// TIA Portal V17 export
// export: Created 2026-04-13T11:12:45.2431947Z, ExportSetting WithDefaults, DisplayName Totally Integrated Automation Portal, DisplayVersion V17 Update 4, DisplayName TIA Portal Openness, DisplayVersion V17 Update 4, DisplayName TIA Portal Version Control Interface, DisplayVersion V17, DisplayName SINAMICS Startdrive Advanced, DisplayVersion V17, DisplayName SINAMICS Startdrive G130, G150, S120, S150, SINAMICS MV, S210, DisplayVersion V17, DisplayName SINAMICS Startdrive G110M, G120, G120C, G120D, G120P, G115D, DisplayVersion V17, DisplayName STEP 7 Professional, DisplayVersion V17 Update 4, DisplayName STEP 7 Safety, DisplayVersion V17, DisplayName WinCC Professional, DisplayVersion V17 Update 4
VAR_GLOBAL   // PLC tag table "IO"
   "I0.0" AT %I0.0 : Bool;
   "I0.1" AT %I0.1 : Bool;
   "I0.2" AT %I0.2 : Bool;
   "I0.3" AT %I0.3 : Bool;
   "I0.4" AT %I0.4 : Bool;
   "I0.5" AT %I0.5 : Bool;
   "I0.6" AT %I0.6 : Bool;
   "I0.7" AT %I0.7 : Bool;
   "I1.0" AT %I1.0 : Bool;
   "I1.1" AT %I1.1 : Bool;
   "I2.0" AT %I2.0 : Bool;
   "I2.1" AT %I2.1 : Bool;
   "I2.2" AT %I2.2 : Bool;
   "I2.3" AT %I2.3 : Bool;
   "I2.4" AT %I2.4 : Bool;
   "I2.5" AT %I2.5 : Bool;
   "I2.6" AT %I2.6 : Bool;
   "I2.7" AT %I2.7 : Bool;
   "I3.0" AT %I3.0 : Bool;
   "I3.1" AT %I3.1 : Bool;
   "I3.2" AT %I3.2 : Bool;
   "I3.3" AT %I3.3 : Bool;
   "I3.4" AT %I3.4 : Bool;
   "I3.5" AT %I3.5 : Bool;
   "I3.6" AT %I3.6 : Bool;
   "I3.7" AT %I3.7 : Bool;
   "I4.0" AT %I4.0 : Bool;
   "I4.1" AT %I4.1 : Bool;
   "I4.2" AT %I4.2 : Bool;
   "I4.3" AT %I4.3 : Bool;
   "I4.4" AT %I4.4 : Bool;
   "I4.5" AT %I4.5 : Bool;
   "I4.6" AT %I4.6 : Bool;
   "I4.7" AT %I4.7 : Bool;
   "I5.0" AT %I5.0 : Bool;
   "I5.1" AT %I5.1 : Bool;
   "I5.2" AT %I5.2 : Bool;
   "I5.3" AT %I5.3 : Bool;
   "I5.4" AT %I5.4 : Bool;
   "I5.5" AT %I5.5 : Bool;
   "I5.6" AT %I5.6 : Bool;
   "I5.7" AT %I5.7 : Bool;
   "Q0.1" AT %Q0.1 : Bool;
   "Q0.2" AT %Q0.2 : Bool;
   "Q0.3" AT %Q0.3 : Bool;
   "Q0.4" AT %Q0.4 : Bool;
   "Q0.5" AT %Q0.5 : Bool;
   "Q0.6" AT %Q0.6 : Bool;
   "Q0.7" AT %Q0.7 : Bool;
   "Q1.0" AT %Q1.0 : Bool;
   "Q1.1" AT %Q1.1 : Bool;
   "Q1.2" AT %Q1.2 : Bool;
   "Q1.3" AT %Q1.3 : Bool;
   "Q1.4" AT %Q1.4 : Bool;
   "Q1.5" AT %Q1.5 : Bool;
   "Q3.0" AT %Q3.0 : Bool;
   "Q3.1" AT %Q3.1 : Bool;
   "Q3.2" AT %Q3.2 : Bool;
   "Q3.3" AT %Q3.3 : Bool;
   "Q3.4" AT %Q3.4 : Bool;
   "Q3.5" AT %Q3.5 : Bool;
   "Q3.6" AT %Q3.6 : Bool;
   "Q3.7" AT %Q3.7 : Bool;
   "Q4.0" AT %Q4.0 : Bool;
   "Q4.1" AT %Q4.1 : Bool;
   "Q4.2" AT %Q4.2 : Bool;
   "Q4.3" AT %Q4.3 : Bool;
   "Q4.4" AT %Q4.4 : Bool;
   "Q4.5" AT %Q4.5 : Bool;
   "Q4.6" AT %Q4.6 : Bool;
   "Q4.7" AT %Q4.7 : Bool;
   "Q5.0" AT %Q5.0 : Bool;
   "Q5.1" AT %Q5.1 : Bool;
   "Q5.2" AT %Q5.2 : Bool;
   "Q5.3" AT %Q5.3 : Bool;
   "Q5.4" AT %Q5.4 : Bool;
   "Q0.0" AT %Q0.0 : Bool;
   "I1.2" AT %I1.2 : Bool;
   "I1.3" AT %I1.3 : Bool;
   "I1.4" AT %I1.4 : Bool;
   "I1.5" AT %I1.5 : Bool;
   "Q5.5" AT %Q5.5 : Bool;
   "Q1.6" AT %Q1.6 : Bool;
   "Q1.7" AT %Q1.7 : Bool;
   "I1.6" AT %I1.6 : Bool;
   "I1.7" AT %I1.7 : Bool;
   "Q5.6" AT %Q5.6 : Bool;
   "Q5.7" AT %Q5.7 : Bool;
   "Q6.0" AT %Q6.0 : Bool;
   "Q6.1" AT %Q6.1 : Bool;
   "Q6.2" AT %Q6.2 : Bool;
   "Q6.3" AT %Q6.3 : Bool;
   "Q6.4" AT %Q6.4 : Bool;
   "Q6.5" AT %Q6.5 : Bool;
   "Q6.6" AT %Q6.6 : Bool;
   "Q6.7" AT %Q6.7 : Bool;
   "Q7.0" AT %Q7.0 : Bool;
   "Q7.1" AT %Q7.1 : Bool;
   "Q7.2" AT %Q7.2 : Bool;
   "Q7.3" AT %Q7.3 : Bool;
   "Q7.4" AT %Q7.4 : Bool;
   "Q7.5" AT %Q7.5 : Bool;
   "Q7.6" AT %Q7.6 : Bool;
   "Q7.7" AT %Q7.7 : Bool;
   "Q8.0" AT %Q8.0 : Bool;
   "Q8.1" AT %Q8.1 : Bool;
   "Q8.2" AT %Q8.2 : Bool;
   "Q8.3" AT %Q8.3 : Bool;
   "Q8.4" AT %Q8.4 : Bool;
   "Q8.5" AT %Q8.5 : Bool;
   "Q8.6" AT %Q8.6 : Bool;
   "Q8.7" AT %Q8.7 : Bool;
   "Q9.0" AT %Q9.0 : Bool;
   "Q9.1" AT %Q9.1 : Bool;
   "Q9.2" AT %Q9.2 : Bool;
   "Q9.3" AT %Q9.3 : Bool;
   "Q9.4" AT %Q9.4 : Bool;
   "Q9.5" AT %Q9.5 : Bool;
   "Q9.6" AT %Q9.6 : Bool;
   "Q9.7" AT %Q9.7 : Bool;
   "Q10.0" AT %Q10.0 : Bool;
   "Q10.1" AT %Q10.1 : Bool;
   "Q10.2" AT %Q10.2 : Bool;
   "Q10.3" AT %Q10.3 : Bool;
   "I6.0" AT %I6.0 : Bool;
   "I6.1" AT %I6.1 : Bool;
   "I6.2" AT %I6.2 : Bool;
   "I6.3" AT %I6.3 : Bool;
   "I6.4" AT %I6.4 : Bool;
   "I6.5" AT %I6.5 : Bool;
   "I6.6" AT %I6.6 : Bool;
   "I6.7" AT %I6.7 : Bool;
   "I7.0" AT %I7.0 : Bool;
   "I7.1" AT %I7.1 : Bool;
   "I7.2" AT %I7.2 : Bool;
   "I7.3" AT %I7.3 : Bool;
   "I7.4" AT %I7.4 : Bool;
   "I7.5" AT %I7.5 : Bool;
   "I7.6" AT %I7.6 : Bool;
   "I7.7" AT %I7.7 : Bool;
   "Q10.4" AT %Q10.4 : Bool;
   "Q10.5" AT %Q10.5 : Bool;
   "Q10.6" AT %Q10.6 : Bool;
   "Q10.7" AT %Q10.7 : Bool;
   "Q11.0" AT %Q11.0 : Bool;
   "Q11.1" AT %Q11.1 : Bool;
   "Q11.2" AT %Q11.2 : Bool;
   "Q11.3" AT %Q11.3 : Bool;
   "Q11.4" AT %Q11.4 : Bool;
   "Q11.5" AT %Q11.5 : Bool;
   "Q11.6" AT %Q11.6 : Bool;
   "Q11.7" AT %Q11.7 : Bool;
   "Q12.0" AT %Q12.0 : Bool;
   "Q12.1" AT %Q12.1 : Bool;
   "Q12.2" AT %Q12.2 : Bool;
   "Q12.3" AT %Q12.3 : Bool;
   "Q12.4" AT %Q12.4 : Bool;
   "Q12.5" AT %Q12.5 : Bool;
   "Q12.6" AT %Q12.6 : Bool;
   "Q12.7" AT %Q12.7 : Bool;
   "Q13.0" AT %Q13.0 : Bool;
   "Q13.1" AT %Q13.1 : Bool;
   "Q13.2" AT %Q13.2 : Bool;
   "Q13.3" AT %Q13.3 : Bool;
   "Q13.4" AT %Q13.4 : Bool;
   "Q13.5" AT %Q13.5 : Bool;
   "Q13.6" AT %Q13.6 : Bool;
   "Q13.7" AT %Q13.7 : Bool;
   "Q14.0" AT %Q14.0 : Bool;
   "Q14.1" AT %Q14.1 : Bool;
   "Q14.2" AT %Q14.2 : Bool;
   "Q14.3" AT %Q14.3 : Bool;
   "Q14.4" AT %Q14.4 : Bool;
   "Q14.5" AT %Q14.5 : Bool;
   "Q14.6" AT %Q14.6 : Bool;
   "Q14.7" AT %Q14.7 : Bool;
   "Q15.0" AT %Q15.0 : Bool;
   "Q15.1" AT %Q15.1 : Bool;
   "Q15.2" AT %Q15.2 : Bool;
   "Q15.3" AT %Q15.3 : Bool;
   "Q15.4" AT %Q15.4 : Bool;
   "Q15.5" AT %Q15.5 : Bool;
   "Q15.6" AT %Q15.6 : Bool;
   "Q15.7" AT %Q15.7 : Bool;
   "Q16.0" AT %Q16.0 : Bool;
   "Q16.1" AT %Q16.1 : Bool;
   "Q16.2" AT %Q16.2 : Bool;
   "Q16.3" AT %Q16.3 : Bool;
   "Q16.4" AT %Q16.4 : Bool;
   "Q16.5" AT %Q16.5 : Bool;
   "Q16.6" AT %Q16.6 : Bool;
   "Q16.7" AT %Q16.7 : Bool;
   "Q17.0" AT %Q17.0 : Bool;
   "Q17.1" AT %Q17.1 : Bool;
   "Q17.2" AT %Q17.2 : Bool;
   "Q17.3" AT %Q17.3 : Bool;
   "Q17.4" AT %Q17.4 : Bool;
   "Q17.5" AT %Q17.5 : Bool;
   "Q17.6" AT %Q17.6 : Bool;
   "Q17.7" AT %Q17.7 : Bool;
   "Q18.0" AT %Q18.0 : Bool;
   "Q18.1" AT %Q18.1 : Bool;
   "Q18.2" AT %Q18.2 : Bool;
   "Q18.3" AT %Q18.3 : Bool;
   "Q18.4" AT %Q18.4 : Bool;
   "Q18.5" AT %Q18.5 : Bool;
   "Q18.6" AT %Q18.6 : Bool;
   "Q18.7" AT %Q18.7 : Bool;
   "Q19.0" AT %Q19.0 : Bool;
   "Q19.1" AT %Q19.1 : Bool;
   "Q19.2" AT %Q19.2 : Bool;
   "Q19.3" AT %Q19.3 : Bool;
   "Q19.4" AT %Q19.4 : Bool;
   "Q19.5" AT %Q19.5 : Bool;
   "Q19.6" AT %Q19.6 : Bool;
   "Q19.7" AT %Q19.7 : Bool;
   "Q20.0" AT %Q20.0 : Bool;
   "Q20.1" AT %Q20.1 : Bool;
   "Q20.2" AT %Q20.2 : Bool;
   "Q20.3" AT %Q20.3 : Bool;
   "Q20.4" AT %Q20.4 : Bool;
   "Q20.5" AT %Q20.5 : Bool;
   "Q2.0" AT %Q2.0 : Bool;
   "Q2.1" AT %Q2.1 : Bool;
   "Q2.2" AT %Q2.2 : Bool;
   "Q2.3" AT %Q2.3 : Bool;
   "Q2.4" AT %Q2.4 : Bool;
   "Q2.5" AT %Q2.5 : Bool;
   "Q2.6" AT %Q2.6 : Bool;
   "Q2.7" AT %Q2.7 : Bool;
END_VAR
